(* CODESYS project sequencia.project

Project tree, tasks and I/O mapping:
  Device : CODESYS Control Win V3, 3S - Smart Software Solutions GmbH, order no. 305021, version 3.5.11.30
    application Application
      libraries: Standard, * (System)
      task MainTask (cyclic, interval t#20ms, priority 1) calls PLC_PRG
      program PLC_PRG [ST]
      function block FBSequencia [ST]
*)

// Device/Application/PLC_PRG
PROGRAM PLC_PRG
VAR
	sinal : REAL;
	saida : ARRAY [0..3] OF BOOL;
	inval : ARRAY [0..3] OF REAL := [0, 0.5, 1, 1.5];
	Seq1 : FBSequencia;
	Seq2 : FBSequencia;
	Seq3 : FBSequencia;
	Seq4 : FBSequencia;
END_VAR

Seq1(invalue:=sinal,desini:=inval[0], outd=>saida[0]);
Seq2(invalue:=sinal,desini:=inval[1], outd=>saida[1]);
Seq3(invalue:=sinal,desini:=inval[2], outd=>saida[2]);
Seq4(invalue:=sinal,desini:=inval[3], outd=>saida[3]);

END_PROGRAM

// Device/Application/FBSequencia
FUNCTION_BLOCK FBSequencia
VAR_INPUT
	invalue:REAL;
	desini: REAL;
END_VAR

VAR_OUTPUT
	outd : BOOL;
END_VAR

VAR
	cicloOn: REAL := 1;
	cicloOf: REAL := 1;
	lowlimit: REAL;
	hilimit: REAL;
	i: INT;
END_VAR

lowlimit :=desini;

i:=0;

FOR i:=0 TO 5 DO
	hilimit := lowlimit + cicloOn;
	IF (invalue >= lowlimit) AND (invalue <= hilimit) THEN
		outd:=TRUE;
		EXIT;
	ELSE 
		outd:=FALSE;
	END_IF
	lowlimit:=hilimit+cicloOf;
END_FOR

END_FUNCTION_BLOCK
